(* PLC project CoDeSys External Library Template, WAGO e!COCKPIT e!COCKPIT, author 3S - Smart Software Solutions GmbH *)
(* stored: creationDateTime 2019-10-29T12:22:40.8044438, version 3.5.5.30, modificationDateTime 2019-10-24T14:40:07.960949, organization 3S - Smart Software Solutions GmbH *)
(* Library project template with all possible element types, docu and a sample project structure *)

(* funkcja bez parametrów zwracająca STRING z bieżącym czasem UTC *)
FUNCTION fnCzasUTC : alSTRINGKomunikat
  VAR
    sCzasUTC : STRING;  (* zmienna do przechowywania wyniku - czas w formacie UTC *)
    dtDataIGodzina : DT;  (* odczyt daty i godziny z systemu *)
    ltGodzina : LTIME;  (* odczyt ms z systemu *)
    sDataiGodzina : STRING;  (* odczyt daty i godziny z systemu - konwersja na STRING *)
    sGodzina : STRING;  (* odczyt ms z systemu - konwersjan a STRING *)
    xMsZapisane : BOOL;  (* flaga informująca czy ms zostały już dopisane *)
  END_VAR

            (*odczyt czasu z systemu i jego konwersja do STRING*)

dtDataIGodzina := FuGetDateAndTime();
ltGodzina := FuGetLongTime();
sDataiGodzina := DT_TO_STRING(dtDataiGodzina);
sGodzina := LTIME_TO_STRING(ltGodzina);

sCzasUTC := MID(sDataIGodzina , 4 , 4);							(*dodanie roku do wyniku*)
sCzasUTC := CONCAT(sCzasUTC , '-');
sCzasUTC := CONCAT(sCzasUTC , MID(sDataIGodzina , 2 , 9));		(*dodanie miesiąca do wyniku*)
sCzasUTC := CONCAT(sCzasUTC , '-');
sCzasUTC := CONCAT(sCzasUTC , MID(sDataIGodzina , 2 , 12));		(*dodanie dnia do wyniku*)
sCzasUTC := CONCAT(sCzasUTC , 'T');
sCzasUTC := CONCAT(sCzasUTC , MID(sDataIGodzina , 2 , 15));		(*dodanie godziny do wyniku*)
sCzasUTC := CONCAT(sCzasUTC , ':');
sCzasUTC := CONCAT(sCzasUTC , MID(sDataIGodzina , 2 , 18));		(*dodanie minuty do wyniku*)
sCzasUTC := CONCAT(sCzasUTC , ':');
sCzasUTC := CONCAT(sCzasUTC , MID(sDataIGodzina , 2 , 21));		(*dodanie sekundy do wyniku*)
sCzasUTC := CONCAT(sCzasUTC , '.');

(*sprawdzenie czy w danych o czasie są milisekundy*)

IF FIND(sGodzina , 'ms') <> 0 THEN 

	xMsZapisane := FALSE;

(*jeżeli przed wykrytym 'ms' dwa znaki wcześniej nie ma liczby dopisz dwa zera i liczbę jednocyfrową przed 'ms'*)
		
	IF STRING_TO_INT(MID(sGodzina , 1 , FIND(sGodzina , 'ms') - 2)) = 0 AND MID(sGodzina , 1 , FIND(sGodzina , 'ms') - 2) <> '0' AND xMsZapisane = FALSE THEN
		sCzasUTC := CONCAT(sCzasUTC , '00');
		sCzasUTC := CONCAT(sCzasUTC , MID(sGodzina , 1 , FIND(sGodzina , 'ms') - 1));
		xMsZapisane := TRUE;
	END_IF

(*jeżeli przed wykrytym 'ms' trzy znaki wcześniej nie ma liczby dopisz jedno zero i liczbę dwujcyfrową przed 'ms'*)
		
	IF STRING_TO_INT(MID(sGodzina , 1 , FIND(sGodzina , 'ms') - 3)) = 0 AND MID(sGodzina , 1 , FIND(sGodzina , 'ms') - 3) <> '0' AND xMsZapisane = FALSE THEN
		sCzasUTC := CONCAT(sCzasUTC , '0');
		sCzasUTC := CONCAT(sCzasUTC , MID(sGodzina , 2 , FIND(sGodzina , 'ms') - 2));
		xMsZapisane := TRUE;	
	END_IF

(*jeżeli przed wykrytym 'ms' cztery znaki wcześniej nie ma liczby dopisz liczbę trzycyfrową cyfrową przed 'ms'*)

	IF STRING_TO_INT(MID(sGodzina , 1 , FIND(sGodzina , 'ms') - 4)) = 0 AND MID(sGodzina , 1 , FIND(sGodzina , 'ms') - 4) <> '0' AND xMsZapisane = FALSE THEN
		sCzasUTC := CONCAT(sCzasUTC , MID(sGodzina , 3 , FIND(sGodzina , 'ms') - 3));			
	END_IF
		
	ELSE

(*jeżeli nie wykryto 'ms' dopisz trzy zera*)

	sCzasUTC := CONCAT(sCzasUTC , '000');

END_IF

sCzasUTC := CONCAT(sCzasUTC , '+00:00');

fnCzasUTC :=sCzasUTC;
          
END_FUNCTION
